FUNCTION_BLOCK Links
VAR
	links : Dictionary;
END_VAR

METHOD PUBLIC DisposeAndRemoveAll
VAR
	enumerator : I_ForwardEnumerator;
	currentLink : I_Link;
END_VAR
enumerator := links.GetEnumerator();

WHILE (enumerator.MoveNext()) DO
	IF enumerator.TryGet(currentLink) THEN
		currentLink.Dispose();
	END_IF
END_WHILE

enumerator.Dispose();
links.Clear();
END_METHOD

METHOD PUBLIC GetById : I_Link
VAR_INPUT
	Id : T_MAXSTRING;
END_VAR
links.TryGetValue(Id,GetById);
END_METHOD

METHOD PUBLIC Insert
VAR_INPUT
	Link : I_Link;
END_VAR
IF Link = 0 THEN
	RETURN;
END_IF

links.AddOrUpdate(Link.Id,Link);
END_METHOD

END_FUNCTION_BLOCK

(* stored: Version 1.1.0.1, ProductVersion 3.1.4024.12
   POU Links: Id {827eb88a-80de-000d-1d2f-a85a6f23f332}, SpecialFunc None
   Method DisposeAndRemoveAll: Id {0d394ea8-a653-0e33-368b-b6719124cb4f}
   Method GetById: Id {c399e1f7-8497-0d5f-150c-9d7b13ed5610}
   Method Insert: Id {1b2ad055-14f8-0fec-371f-f33113ebd2b6} *)
